// TwinCAT 3 PLC project test_lv0
// ProgramVersion: 3.1.4020.1
// libraries:
//   Tc2_Standard, * (Beckhoff Automation GmbH)
//   Tc2_System, * (Beckhoff Automation GmbH)
//   Tc3_Module, * (Beckhoff Automation GmbH)
//   tclib_ph_lv0, * (Poh)
// project tree:
//   / GlobalTextList.TcGTLO, PlcTask.TcTTO
//   POUs/ MAIN.TcPOU, Visualization.TcVIS
// (motion and I/O tree: see PLC project ph_lv0)
// real-time tasks:
//   TASK PlcTask: cycle T#10ms, priority 20, ADS port 350
// variable links:

CONFIGURATION test_lv0
    RESOURCE PLC ON TwinCAT3
        TASK PlcTask(INTERVAL := T#10ms, PRIORITY := 20);
        PROGRAM MAIN WITH PlcTask : MAIN;
    END_RESOURCE
END_CONFIGURATION

// ---- POUs/MAIN.TcPOU
PROGRAM MAIN
VAR
	m_tg_OnOff : M_TRIGGERS;
	State : INT := -10;
	bSignal : BOOL;
	Rise_Count, Fall_Count, RiseFall_Count : INT := 0;
	t_Rise_Count, t_Fall_Count, t_RiseFall_Count : INT := 0;
	m_trigger_test_ok : BOOL := FALSE;
END_VAR

m_trigger_test();

ACTION m_trigger_test:
m_tg_OnOff(BOOL_IN:= bSignal, BOOL_R=> , BOOL_F=> , BOOL_RF=> );

IF m_tg_OnOff.BOOL_R THEN
	Rise_Count := Rise_Count + 1;
END_IF
IF m_tg_OnOff.BOOL_F THEN
	Fall_Count := Fall_Count + 1;
END_IF
IF m_tg_OnOff.BOOL_RF THEN
	RiseFall_Count := RiseFall_Count + 1;
END_IF

CASE State OF 
0: 
	m_trigger_test_ok := FALSE;
	bSignal := FALSE;	
	Rise_Count := 0;
 	Fall_Count := 0; 
	RiseFall_Count := 0;
	t_Rise_Count := 0;
 	t_Fall_Count := 0; 
	t_RiseFall_Count := 0;
	State := State + 1;
1:
	bSignal := TRUE;
	State := State + 1;
2:
	IF Rise_Count <> t_Rise_Count AND RiseFall_Count <> t_RiseFall_Count THEN
		t_Rise_Count := Rise_Count;
		t_Fall_Count := Fall_Count; 
		t_RiseFall_Count := RiseFall_Count;
		State := State + 1;
	END_IF
3:
	bSignal := FALSE;
	State := State + 1;
4: 
	IF Fall_Count <> t_Fall_Count AND RiseFall_Count <> t_RiseFall_Count THEN
		t_Rise_Count := Rise_Count;
		t_Fall_Count := Fall_Count; 
		t_RiseFall_Count := RiseFall_Count;
		State := State + 1;
	END_IF
5:
	m_trigger_test_ok := TRUE;
	State := -10;
END_CASE
END_ACTION

END_PROGRAM

// ---- POUs/Visualization.TcVIS
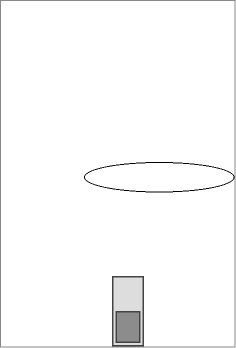
VISUALIZATION Visualization  // 236x348
    Ellipse (84,162 150x30)
    DipSwitch (93,276 70x70), variable: MAIN.bSignal, behaviour: TOGGLE, style: Switch-DipSwitch-Gray
END_VISUALIZATION
